PROGRAM control
VAR
	driverModeVar	: INT :=1;
	driverMode1		: BOOL;
	driverMode2		: BOOL;
	driverMode3		: BOOL;
	invisibleGUI	: BOOL := FALSE;
	visibleGUI		: BOOL := FALSE;
END_VAR

//Laitteen tilan asetus:
CASE GVL.driverMode OF
	1:	IF GVL.start AND NOT(GVL.vikamuisti) THEN
			GVL.systemOn := TRUE;
			driverModeVar := GVL.driverMode;
		END_IF
		IF NOT(GVL.safetyOk) OR GVL.stop THEN
			GVL.systemOn := FALSE;
		END_IF
		
		IF NOT(GVL.safetyOk) THEN
			GVL.vikamuisti := TRUE;
		END_IF
		IF GVL.reset THEN
			GVL.vikamuisti := FALSE;
		END_IF
		
	2:	IF GVL.startGUI AND NOT(GVL.vikamuisti) THEN
			GVL.systemOn := TRUE;
			driverModeVar := GVL.driverMode;
		END_IF
		IF NOT(GVL.safetyOk) OR GVL.stopGUI THEN
			GVL.systemOn := FALSE;
		END_IF
		
		IF NOT(GVL.safetyOk) THEN
			GVL.vikamuisti := TRUE;
		END_IF
		IF GVL.resetGUI THEN
			GVL.vikamuisti := FALSE;
		END_IF
		
	3:	IF GVL.startGUI AND NOT(GVL.vikamuisti) THEN
			GVL.systemOn := TRUE;
			driverModeVar := GVL.driverMode;
		END_IF
		IF NOT(GVL.safetyOk) OR GVL.stopGUI THEN
			GVL.systemOn := FALSE;
		END_IF		
END_CASE

IF driverModeVar <> GVL.driverMode THEN
	GVL.systemOn := FALSE;
END_IF

IF GVL.driverMode = 3 THEN
	invisibleGUI := TRUE;
	visibleGUI := FALSE;
ELSE
	invisibleGUI := FALSE;
	visibleGUI := TRUE; 
END_IF

//IF GVL.start THEN
//	driverModeVar := GVL.driverMode;
//END_IF

IF GVL.tila1 AND NOT(GVL.tila2) THEN
	GVL.driverMode := 1;
	driverMode1 := FALSE;
ELSE
	driverMode1 := TRUE;
END_IF

IF NOT(GVL.tila2) AND NOT(GVL.tila1) THEN
	GVL.driverMode := 2;
	driverMode2 := FALSE;
ELSE
	driverMode2 := TRUE;
END_IF

IF NOT(GVL.tila1) AND GVL.tila2 THEN
	GVL.driverMode := 3;
	driverMode3 := FALSE;
ELSE
	driverMode3 := TRUE;
END_IF

END_PROGRAM

(* stored: Version 1.1.0.1, ProductVersion 3.1.4024.11
   POU control: Id {f4192589-e639-46b2-82cf-0b85b345678c}, SpecialFunc None *)
